PROGRAM MAIN
VAR
	i: INT;
END_VAR

i:=i+1;

END_PROGRAM

(* stored: Version 1.1.0.1, ProductVersion 3.1.4024.4
   POU MAIN: Id {b193803e-6fed-4b21-a10d-aaf3d7cf5720}, SpecialFunc None *)
